PROGRAM MAIN
VAR
	eLedColor				:E_Color;
	i						:INT;
	bLed1			AT %Q*	:ARRAY[E_Color.eRed..E_Color.eWhite] OF BOOL;
	bLed2			AT %Q*	:ARRAY[E_Color.eRed..E_Color.eWhite] OF BOOL;
END_VAR

i:=i+1;

IF i=10 THEN
	bLed1[E_Color.eRed]:=TRUE;
ELSIF i=20 THEN
	bLed1[E_Color.eYellow]:=TRUE;
ELSIF i=30 THEN
	bLed1[E_Color.eGreen]:=TRUE;
ELSIF i=40 THEN
	bLed1[E_Color.eWhite]:=TRUE;
ELSIF i=50 THEN
	bLed2[E_Color.eRed]:=TRUE;
ELSIF i=60 THEN
	bLed2[E_Color.eYellow]:=TRUE;
ELSIF i=70 THEN
	bLed2[E_Color.eGreen]:=TRUE;
ELSIF i=80 THEN
	bLed2[E_Color.eWhite]:=TRUE;
ELSIF i=100 THEN
	FOR eLedColor:= E_Color.eRed TO E_Color.eWhite DO
		bLed1[eLedColor]:=FALSE;
		bLed2[eLedColor]:=FALSE;
	END_FOR
	i:=0;
END_IF

END_PROGRAM

(* stored: Version 1.1.0.1
   POU MAIN: Id {4224c9ea-319d-4468-8ed0-878cb34713a5}, SpecialFunc None *)
